Fanuc KAREL source: kt00487.KL

PROGRAM KT00487
%STACKSIZE=65535
%PRIORITY=65535
%NOLOCKGROUP
VAR
P1 : POSITION
P2 : XYZWPREXT
OUT : JOINTPOS9
BEGIN
P2.Y=2.0
-- UNRESOLVED_PC line 9 opcodes [49 49 7E 60 7E 4A] marker_code=20
END KT00487
